// TwinCAT 3 PLC project PKE_Graz
// ProgramVersion: 3.1.4023.0
// libraries:
//   EfficientIO Communicator, * (EfficientIO)
//   Lynus Energy Basic, * (Lynus AG)
//   Lynus Energy ModbusTCP, * (Lynus AG)
//   Lynus Persistent Data V1, * (Lynus AG)
//   Lynus Standards, * (Lynus AG)
//   Tc2_ModbusSrv, * (Beckhoff Automation GmbH)
//   Tc2_Standard, * (Beckhoff Automation GmbH)
//   Tc2_System, * (Beckhoff Automation GmbH)
//   Tc2_Utilities, * (Beckhoff Automation GmbH)
//   Tc3_Module, * (Beckhoff Automation GmbH)
// project tree:
//   / FastTask.TcTTO, MiddleTask.TcTTO, SlowTask.TcTTO
//   FB/ FB_ModBus_100Reg_once_FC3.TcPOU, FB_ModBus_2Registers_FC3_T.TcPOU, F_DWORD_TO_FLOAT32.TcPOU
//   POUs/ prgComEffIO.TcPOU, PrgModbus.TcPOU, prgPersistent.TcPOU, prgRWEffIO.TcPOU, prgVarEffIO.TcPOU (not stored)
// real-time tasks:
//   TASK MiddleTask: cycle T#10ms, priority 20, ADS port 350
//   TASK FastTask: cycle T#5ms, priority 19, ADS port 351
//   TASK SlowTask: cycle T#20ms, priority 21, ADS port 352

CONFIGURATION PKE_Graz
    RESOURCE PLC ON TwinCAT3
        TASK FastTask(INTERVAL := T#5ms, PRIORITY := 19);
        TASK MiddleTask(INTERVAL := T#10ms, PRIORITY := 20);
        TASK SlowTask(INTERVAL := T#20ms, PRIORITY := 21);
        PROGRAM prgRWEffIO WITH FastTask : prgRWEffIO;
        PROGRAM prgVarEffIO WITH FastTask : prgVarEffIO;
        PROGRAM prgPersistent WITH MiddleTask : prgPersistent;
        PROGRAM PrgModbus WITH MiddleTask : PrgModbus;
        PROGRAM prgComEffIO WITH SlowTask : prgComEffIO;
    END_RESOURCE
END_CONFIGURATION

// ---- POUs/prgRWEffIO.TcPOU
PROGRAM prgRWEffIO
VAR
	fbRW1		: FB_ReadWrite_V2;
END_VAR

fbRW1(	eUploadType := eSelectDataUploadType.e_Change_Intervall5min,
		bBusy=> , 
		bError=> , 
		udiErrorCodeOut=> , 
		eErrorReadWrite_Out=> );

END_PROGRAM

// ---- POUs/prgPersistent.TcPOU
PROGRAM prgPersistent
VAR
	fbUSV		: FB_WritePersistentData_General;
	
	fb_Reboot		: NT_reboot;
	m_Reboot		: BOOL:=FALSE;
END_VAR

fbUSV(
	eSaveModeData:= eUSVSaveMode.eSaveEventBased, 
	bLoadPersistentDataOk=> , 
//	bPowerFailDetect=> , 
	bError=> , 
	bySaveProcess=> , 
	dwStorageLast24h=> , 
	udiErrorCode=> );
	
	
fb_Reboot(	netid := '',
			delay := 2,
			start := m_Reboot);

END_PROGRAM

// ---- POUs/PrgModbus.TcPOU
PROGRAM PrgModbus
VAR
	FB_Modbus: FB_ModBus_100Reg_once_FC3;
	fb_MB_WatchDog:FB_MBWriteSingleCoil ;
	fb_MB_Multi: FB_MBWriteRegs;

	str_IP	:STRING(20);
	
	i: INT;
	i_State: INT;
	ton_Wait_time: Ton;
	ton_TimeOut: ton;
	w_Array_Received: ARRAY [0..450] OF WORD;

	w_Array_Pol1_1: ARRAY [0..99] OF WORD;
	m_Pol1_1_ok: BOOL;
	w_Array_Pol1_2: ARRAY [0..99] OF WORD;
	m_Pol1_2_ok: BOOL;
	w_Array_Pol1_3: ARRAY [0..99] OF WORD;
	m_Pol1_3_ok: BOOL;
	w_Array_Pol1_4: ARRAY [0..99] OF WORD;
	m_Pol1_4_ok: BOOL;
	w_Array_Pol1_5: ARRAY [0..99] OF WORD;
	m_Pol1_5_ok: BOOL;
	w_Array_Pol1_6: ARRAY [0..99] OF WORD;
	m_Pol1_6_ok: BOOL;	
	int_Timeout: ARRAY [1..6] OF INT;
	
	real_EG_0_01_Testraum_Temp	: REAL;										//{#lynus.ag#()}
	real_EG_0_02_Werkstatt_Temp	: REAL;										//{#lynus.ag#()}
	real_EG_0_04_Buero1_Temp	: REAL;										//{#lynus.ag#()}
	real_EG_0_05_Buero2_Temp	: REAL;										//{#lynus.ag#()}
	real_EG_0_06_Leitung_Temp	: REAL;										//{#lynus.ag#()}
	real_EG_0_07_Service_Annahme_Temp	: REAL;								//{#lynus.ag#()}
	real_EG_0_08_Buero3_Temp	: REAL;										//{#lynus.ag#()}
	real_EG_0_09_Buero4_Temp	: REAL;										//{#lynus.ag#()}
	real_EG_0_10_Buero5_Temp	: REAL;										//{#lynus.ag#()}
	real_EG_0_11_Buero6_Temp	: REAL;										//{#lynus.ag#()}
	real_EG_0_12_Buero7_Temp	: REAL;										//{#lynus.ag#()}
	real_EG_0_13_Buero8_Temp	: REAL;										//{#lynus.ag#()}
	real_EG_0_14_Archiv_Temp	: REAL;										//{#lynus.ag#()}
	real_EG_0_20_WC_Damen_Beh_Temp	: REAL;									//{#lynus.ag#()}
	real_EG_0_23_CAD_Reserve_Temp	: REAL;									//{#lynus.ag#()}
	real_EG_0_24_CAD_Temp	: REAL;											//{#lynus.ag#()}
	real_EG_0_25_Reserve_Temp	: REAL;										//{#lynus.ag#()}
	real_EG_0_26_Buero9_Temp	: REAL;										//{#lynus.ag#()}
	real_EG_0_27_ErschliessungEGSued_Temp	: REAL;							//{#lynus.ag#()}
	real_EG_0_27_Teekueche_Temp	: REAL;										//{#lynus.ag#()}
	real_EG_0_28_Buero8_Temp	: REAL;										//{#lynus.ag#()}
	real_EG_0_29_Buero10_Temp	: REAL;										//{#lynus.ag#()}
	real_EG_0_30_Demo_Temp	: REAL;											//{#lynus.ag#()}
	real_EG_0_31_Buero11_Temp	: REAL;										//{#lynus.ag#()}
	real_EG_0_32_Buero12_GF_Temp	: REAL;									//{#lynus.ag#()}
	real_EG_0_33_Buero13_GF_Temp	: REAL;									//{#lynus.ag#()}
	real_EG_0_35_Buero14_Temp	: REAL;										//{#lynus.ag#()}
	real_EG_0_36_Buero15_Temp	: REAL;										//{#lynus.ag#()}
	real_EG_0_37_Buero16_Temp	: REAL;										//{#lynus.ag#()}
	real_EG_0_39_Buero17_Temp	: REAL;										//{#lynus.ag#()}
	real_EG_0_40_Besprechung_Temp	: REAL;									//{#lynus.ag#()}
	real_EG_0_42_WC_Beh_Temp	: REAL;										//{#lynus.ag#()}
	real_H_0_02_LagerPKE_Temp	: REAL;										//{#lynus.ag#()}
	real_H_00_03_Buero_LagerPKE_Temp	: Real;								//{#lynus.ag#()}
	real_OG1_1_01_Empfang_Temp	: REAL;										//{#lynus.ag#()}
	real_OG1_1_03_Buero1_Temp	: REAL;										//{#lynus.ag#()}
	real_OG1_1_04_Buero2_Temp	: REAL;										//{#lynus.ag#()}
	real_OG1_1_05_Buero3_Temp	: REAL;										//{#lynus.ag#()}
	real_OG1_1_06_Buero4_Temp	: REAL;										//{#lynus.ag#()}
	real_OG1_1_07_Buero_Besprechung_Temp	: REAL;							//{#lynus.ag#()}
	real_OG1_1_1_08_Plotter_Temp	: REAL;									//{#lynus.ag#()}
	real_OG1_1_04_WC_Herren_Temp	: REAL;									//{#lynus.ag#()}
	real_OG1_Serverraum_Temp	: REAL;										//{#lynus.ag#()}
	real_OG1_4_01_Empfang_Temp	: REAL;										//{#lynus.ag#()}
	real_OG1_4_03_Lager_Temp	: REAL;										//{#lynus.ag#()}
	real_OG1_4_04_Buero1_Temp	: REAL;										//{#lynus.ag#()}
	real_OG1_4_05_Buero2_Temp	: REAL;										//{#lynus.ag#()}
	real_OG1_4_06_Buero3_Temp	: REAL;										//{#lynus.ag#()}
	real_OG1_4_07_Buero4_Temp	: REAL;										//{#lynus.ag#()}
	real_OG1_4_08_Buero5_Temp	: REAL;										//{#lynus.ag#()}
	real_OG1_4_09_Buero6_Temp	: REAL;										//{#lynus.ag#()}
	real_OG1_4_10_AufenthaltKueche_Temp	: Real;								//{#lynus.ag#()}
	real_OG1_4_11_Besprechung_Temp	: REAL;									//{#lynus.ag#()}
	real_OG1_4_14_WC_Damen_Temp	: REAL;										//{#lynus.ag#()}
	real_OG1_2_03_Buero2_Temp	: REAL;										//{#lynus.ag#()}
	real_OG1_2_04_Besprechung_Temp	: REAL;									//{#lynus.ag#()}
	real_OG1_2_05_Server_VTOG2_Temp	: REAL;									//{#lynus.ag#()}
	real_OG1_2_06_Buero3_Temp	: REAL;										//{#lynus.ag#()}
	real_OG1_2_07_Buero4_Temp	: REAL;										//{#lynus.ag#()}
	real_OG1_3_xx_Besprechung_Temp	: REAL;									//{#lynus.ag#()}
	real_OG1_3_02_Buero1_Temp	: REAL;										//{#lynus.ag#()}
	real_OG1_3_03_Buero2_Temp	: REAL;										//{#lynus.ag#()}
	real_OG1_3_05_Server_Temp	: REAL;										//{#lynus.ag#()}
	real_OG1_3_06_Vorraum_WC_Temp	: REAL;									//{#lynus.ag#()}
	real_OG1_3_09_Empfang_Temp	: REAL;										//{#lynus.ag#()}
	real_OG1_3_10_Buero3_Temp	: REAL;										//{#lynus.ag#()}
	real_OG1_3_11_Buero4_Temp	: REAL;										//{#lynus.ag#()}
	real_H01_VL_Temp	: REAL;												//{#lynus.ag#()}
	real_H01_RL_Temp	: REAL;												//{#lynus.ag#()}
	real_H02_VL_Temp	: REAL;												//{#lynus.ag#()}
	real_H02_RL_Temp	: REAL;												//{#lynus.ag#()}
	real_H03_VL_Temp	: REAL;												//{#lynus.ag#()}
	real_H03_RL_Temp	: REAL;												//{#lynus.ag#()}
	real_H04_VL_Temp	: REAL;												//{#lynus.ag#()}
	real_H04_RL_Temp	: REAL;												//{#lynus.ag#()}
	real_H05_VL_Temp	: REAL;												//{#lynus.ag#()}
	real_H05_RL_Temp	: REAL;												//{#lynus.ag#()}
	real_H06_VL_Temp	: REAL;												//{#lynus.ag#()}
	real_H06_RL_Temp	: REAL;												//{#lynus.ag#()}
	real_SP_Schneider_H01_Temp_HZG	: REAL;									//{#lynus.ag#()}
	real_SP_Schneider_H02_Temp_HZG	: REAL;									//{#lynus.ag#()}
	real_SP_Schneider_H03_Temp_HZG	: REAL;									//{#lynus.ag#()}
	real_SP_Schneider_H04_Temp_HZG	: REAL;									//{#lynus.ag#()}
	real_SP_Schneider_H05_Temp_HZG	: REAL;									//{#lynus.ag#()}
	real_SP_Schneider_H06_Temp_HZG	: REAL;									//{#lynus.ag#()}
	real_SP_Schneider_H01_Temp_KLG	: REAL;									//{#lynus.ag#()}
	real_SP_Schneider_H02_Temp_KLG	: REAL;									//{#lynus.ag#()}
	real_SP_Schneider_H03_Temp_KLG	: REAL;									//{#lynus.ag#()}
	real_SP_Schneider_H04_Temp_KLG	: REAL;									//{#lynus.ag#()}
	real_SP_Schneider_H05_Temp_KLG	: REAL;									//{#lynus.ag#()}
	real_SP_Schneider_H06_Temp_KLG	: REAL;									//{#lynus.ag#()}
	real_L01_ZUL_Temp	: REAL;												//{#lynus.ag#()}
	real_L01_ABL_Temp	: REAL;												//{#lynus.ag#()}
	real_L01_AUL_Temp	: REAL;												//{#lynus.ag#()}
	real_L01_FOL_Temp	: REAL;												//{#lynus.ag#()}
	real_L01_SE_ZUL_Temp	: REAL;											//{#lynus.ag#()}
	real_L01_SW_Rot_WT	: REAL;												//{#lynus.ag#()}
	real_L01_SW_E_HZ_Reg	: REAL;											//{#lynus.ag#()}
	real_AT	: REAL;															//{#lynus.ag#()}
	real_SP_EfficientIO_H01_Temp_HZG	: Real;								//{#lynus.ag#()}
	real_SP_EfficientIO_H02_Temp_HZG	: Real;								//{#lynus.ag#()}
	real_SP_EfficientIO_H03_Temp_HZG	: Real;								//{#lynus.ag#()}
	real_SP_EfficientIO_H04_Temp_HZG	: Real;								//{#lynus.ag#()}
	real_SP_EfficientIO_H05_Temp_HZG	: Real;								//{#lynus.ag#()}
	real_SP_EfficientIO_H06_Temp_HZG	: Real;								//{#lynus.ag#()}
	real_SP_EfficientIO_H01_Temp_KLG	: Real;								//{#lynus.ag#()}
	real_SP_EfficientIO_H02_Temp_KLG	: Real;								//{#lynus.ag#()}
	real_SP_EfficientIO_H03_Temp_KLG	: Real;								//{#lynus.ag#()}
	real_SP_EfficientIO_H04_Temp_KLG	: Real;								//{#lynus.ag#()}
	real_SP_EfficientIO_H05_Temp_KLG	: Real;								//{#lynus.ag#()}
	real_SP_EfficientIO_H06_Temp_KLG	: Real;								//{#lynus.ag#()}
	real_SP_EfficientIO_H01_Temp_HZG_received	: REAL;				
	real_SP_EfficientIO_H02_Temp_HZG_received	: REAL;				
	real_SP_EfficientIO_H03_Temp_HZG_received	: REAL;				
	real_SP_EfficientIO_H04_Temp_HZG_received	: REAL;				
	real_SP_EfficientIO_H05_Temp_HZG_received	: REAL;				
	real_SP_EfficientIO_H06_Temp_HZG_received	: REAL;				
	real_SP_EfficientIO_H01_Temp_KLG_received	: REAL;				
	real_SP_EfficientIO_H02_Temp_KLG_received	: REAL;				
	real_SP_EfficientIO_H03_Temp_KLG_received	: REAL;				
	real_SP_EfficientIO_H04_Temp_KLG_received	: REAL;				
	real_SP_EfficientIO_H05_Temp_KLG_received	: REAL;				
	real_SP_EfficientIO_H06_Temp_KLG_received	: REAL;				
	usint_Betriebsart_H01	: USINT;										//{#lynus.ag#()}
	usint_Betriebsart_H02	: USINT;										//{#lynus.ag#()}
	usint_Betriebsart_H03	: USINT;										//{#lynus.ag#()}
	usint_Betriebsart_H04	: USINT;										//{#lynus.ag#()}
	usint_Betriebsart_H05	: USINT;										//{#lynus.ag#()}
	usint_Betriebsart_H06	: USINT;										//{#lynus.ag#()}
	m_Watchdog	: BOOL;														//{#lynus.ag#()}
	real_ZUL_errechnet_Schneider_Temp	: Real;								//{#lynus.ag#()}
	real_ZUL_errechnet_EfficientIO_Temp	: Real;								//{#lynus.ag#()}
	real_ZUL_errechnet_EfficientIO_Temp_received : REAL;
	FB_Convert_Real_to_Word:		 FB_CV_REAL_FLOAT_TO_WORD;
	f_trig_BussyWrite: f_trig;
	intArray_WriteError				: ARRAY[1..3] OF INT;		//error counter for each write command
	wArray_Data_To_Send				: ARRAY[1..40] OF WORD;		//word array to write 
	TON_HeartBeat2: Ton;
	TON_HeartBeat1: Ton;
	mEnable: BOOL;
	w_adress: WORD;
	nUnitID: BYTE;
	FB_2Reg :FB_ModBus_2Registers_FC3_T;

	ton_Wait2_time: TON;
	intArray_PollOk:  ARRAY [1..6] OF INT;
	intArray_WriteOk:  ARRAY [1..3] OF INT;

	m_Mode_Off_H01				: BOOL;									//{#lynus.ag#()}
	m_Mode_Heating_H01			: BOOL;									//{#lynus.ag#()}
	m_Mode_ReducedHeating_H01	: BOOL;									//{#lynus.ag#()}
	m_Mode_Frost_H01			: BOOL;									//{#lynus.ag#()}
	m_Mode_Cooling_H01			: BOOL;									//{#lynus.ag#()}
	m_Mode_ReducedCooling_H01	: BOOL;									//{#lynus.ag#()}

	m_Mode_Off_H02				: BOOL;									//{#lynus.ag#()}
	m_Mode_Heating_H02			: BOOL;									//{#lynus.ag#()}
	m_Mode_Frost_H02			: BOOL;									//{#lynus.ag#()}
	m_Mode_Cooling_H02			: BOOL;									//{#lynus.ag#()}

	m_Mode_Off_H03				: BOOL;									//{#lynus.ag#()}
	m_Mode_Heating_H03			: BOOL;									//{#lynus.ag#()}
	m_Mode_Frost_H03			: BOOL;									//{#lynus.ag#()}
	m_Mode_Cooling_H03			: BOOL;									//{#lynus.ag#()}

	m_Mode_Off_H04				: BOOL;									//{#lynus.ag#()}
	m_Mode_Heating_H04			: BOOL;									//{#lynus.ag#()}
	m_Mode_Frost_H04			: BOOL;									//{#lynus.ag#()}
	m_Mode_Cooling_H04			: BOOL;									//{#lynus.ag#()}

	m_Mode_Off_H05				: BOOL;									//{#lynus.ag#()}
	m_Mode_Heating_H05			: BOOL;									//{#lynus.ag#()}
	m_Mode_Frost_H05			: BOOL;									//{#lynus.ag#()}
	m_Mode_Cooling_H05			: BOOL;									//{#lynus.ag#()}

	m_Mode_Off_H06				: BOOL;									//{#lynus.ag#()}
	m_Mode_Heating_H06			: BOOL;									//{#lynus.ag#()}
	m_Mode_Frost_H06			: BOOL;									//{#lynus.ag#()}
	m_Mode_Cooling_H06			: BOOL;									//{#lynus.ag#()}

	
	
	int_HeartBeat					: INT;										//{#lynus.ag#()}
	byte_ErrorWarning				: BYTE;										//{#lynus.ag#()}
	m_EnergyOptimicingReady			: BOOL;										//{#lynus.ag#()}

	real_Power_H01				:REAL;									//{#lynus.ag#()}
	real_Power_H02				:REAL;									//{#lynus.ag#()}
	real_Power_H03				:REAL;									//{#lynus.ag#()}
	real_Power_H04				:REAL;									//{#lynus.ag#()}
	real_Power_H05				:REAL;									//{#lynus.ag#()}
	real_Power_H06				:REAL;									//{#lynus.ag#()}
	
	real_EnergyHeating_H01				:REAL;									//{#lynus.ag#()}
	real_EnergyHeating_H02				:REAL;									//{#lynus.ag#()}
	real_EnergyHeating_H03				:REAL;									//{#lynus.ag#()}
	real_EnergyHeating_H04				:REAL;									//{#lynus.ag#()}
	real_EnergyHeating_H05				:REAL;									//{#lynus.ag#()}
	real_EnergyHeating_H06				:REAL;									//{#lynus.ag#()}

	real_EnergyCooling_H01				:REAL;									//{#lynus.ag#()}
	real_EnergyCooling_H02				:REAL;									//{#lynus.ag#()}
	real_EnergyCooling_H03				:REAL;									//{#lynus.ag#()}
	real_EnergyCooling_H04				:REAL;									//{#lynus.ag#()}
	real_EnergyCooling_H05				:REAL;									//{#lynus.ag#()}
	real_EnergyCooling_H06				:REAL;									//{#lynus.ag#()}
	
	real_Power_HeatPump1				:REAL;									//{#lynus.ag#()}
	real_Power_HeatPump2				:REAL;									//{#lynus.ag#()}
	
	int_Count: INT;
END_VAR
VAR PERSISTENT
	m_EnableHeartbeat: BOOL;												//{#lynus.ag#()}
	m_Enbale_Write: BOOL:=TRUE;
END_VAR

// state maschine modbus
(*
FB_2Reg(
	m_Enable:= mEnable , 
	str_IPAdress:= '10.148.188.27', 
	w_Adress:= w_adress, 
	int_Divider:= 1, 
	n_UnitID:= nUnitID, 
	m_Float32Conversion:= , 
	m_PollSuccessful=> , 
	r_ReceivedValue=> , 
	udint_Error_ID=> );
*)

CASE i_State OF
	0: // wait state
		ton_Wait_time.IN := TRUE;
		IF ton_Wait_time.Q THEN
			ton_Wait_time.IN :=FALSE;
			i_State := 1;
		END_IF
	
	
	1: // Poll 1 Register 200 - 299
		FB_Modbus.m_Enable := TRUE;
		FB_Modbus.w_Adress := 199; //201;
		FB_Modbus.usint_Quantity := 100;
		
		ton_TimeOut.IN := TRUE;
		
		// wait for received values
		IF  FB_Modbus.m_PollSuccessful THEN
			FB_Modbus.m_Enable := FALSE;
			m_Pol1_1_ok := TRUE;			
			w_Array_Pol1_1 := FB_Modbus.w_Array_Received;
			FOR i:=0 TO FB_Modbus.usint_Quantity-1 BY 1 DO
				w_Array_Received[200+i] := w_Array_Pol1_1[i];
				w_Array_Pol1_1[i]:=0;
			END_FOR
			ton_TimeOut.IN := FALSE;
			i_State := 2;
		END_IF
		IF ton_TimeOut.Q THEN
			FB_Modbus.m_Enable := FALSE;
			ton_TimeOut.IN := FALSE;
			m_Pol1_1_ok := FALSE;			
			int_Timeout[1] := int_Timeout[1]+1;
			i_State := 2;
		END_IF
	
	2: // wait one cycle
		IF m_Pol1_1_ok THEN 
			m_Pol1_1_ok := FALSE;
			intArray_PollOk[1]:=intArray_PollOk[1]+1;
		END_IF
		i_State := 3;
		
	3: // Poll 2 Register 300 - 399
		FB_Modbus.m_Enable := TRUE;
		FB_Modbus.w_Adress := 299; //301;
		FB_Modbus.usint_Quantity := 100;
		
		ton_TimeOut.IN := TRUE;
		
		// wait for received values
		IF  FB_Modbus.m_PollSuccessful THEN
			FB_Modbus.m_Enable := FALSE;
			m_Pol1_2_ok := TRUE;
			w_Array_Pol1_2 := FB_Modbus.w_Array_Received;
			FOR i:=0 TO FB_Modbus.usint_Quantity-1 BY 1 DO
				w_Array_Received[300+i] := w_Array_Pol1_2[i];
				w_Array_Pol1_2[i]:=0;
			END_FOR
			ton_TimeOut.IN := FALSE;
			i_State := 4;
		END_IF
		IF ton_TimeOut.Q THEN
			FB_Modbus.m_Enable := FALSE;			
			ton_TimeOut.IN := FALSE;
			m_Pol1_2_ok := FALSE;
			int_Timeout[2] := int_Timeout[2]+1;
			i_State := 4;
		END_IF		
	
	4: // wait one cycle
		IF m_Pol1_2_ok THEN 
			m_Pol1_2_ok := FALSE;
			intArray_PollOk[2]:=intArray_PollOk[2]+1;
		END_IF		
		i_State := 5;
		
	5: // Poll 3 Register 400 - 426
		FB_Modbus.m_Enable := TRUE;
		FB_Modbus.w_Adress := 399; //401;
		FB_Modbus.usint_Quantity := 28;
		
		ton_TimeOut.IN := TRUE;
		
		// wait for received values
		IF  FB_Modbus.m_PollSuccessful THEN
			FB_Modbus.m_Enable := FALSE;
			m_Pol1_3_ok := TRUE;
			w_Array_Pol1_3 := FB_Modbus.w_Array_Received;
			FOR i:=0 TO FB_Modbus.usint_Quantity-1 BY 1 DO
				w_Array_Received[400+i] := w_Array_Pol1_3[i];
				w_Array_Pol1_3[i]:=0;
			END_FOR			
			ton_TimeOut.IN := FALSE;
			i_State := 6;
		END_IF
		IF ton_TimeOut.Q THEN
			FB_Modbus.m_Enable := FALSE;		
			ton_TimeOut.IN := FALSE;
			m_Pol1_3_ok := FALSE;
			int_Timeout[3] := int_Timeout[3]+1;
			i_State := 6;
		END_IF		

	6: // wait one cycle
		IF m_Pol1_3_ok THEN 
			m_Pol1_3_ok := FALSE;
			intArray_PollOk[3]:=intArray_PollOk[3]+1;
		END_IF		
		i_State := 7;
		
	7: // Poll 4 Register 432 - 436
		FB_Modbus.m_Enable := TRUE;
		FB_Modbus.w_Adress := 431; 
		FB_Modbus.usint_Quantity := 4;
		
		ton_TimeOut.IN := TRUE;
		
		// wait for received values
		IF  FB_Modbus.m_PollSuccessful THEN
			FB_Modbus.m_Enable := FALSE;
			m_Pol1_4_ok := TRUE;
			w_Array_Pol1_4 := FB_Modbus.w_Array_Received;
			FOR i:=0 TO FB_Modbus.usint_Quantity-1 BY 1 DO
				w_Array_Received[432+i] := w_Array_Pol1_4[i];
				w_Array_Pol1_4[i]:=0;
			END_FOR			
			ton_TimeOut.IN := FALSE;
			i_State := 8;
		END_IF
		IF ton_TimeOut.Q THEN
			FB_Modbus.m_Enable := FALSE;		
			ton_TimeOut.IN := FALSE;
			m_Pol1_4_ok := FALSE;
			int_Timeout[4] := int_Timeout[4]+1;
			i_State := 8;
		END_IF		
		
	8: // wait one cycle
		IF m_Pol1_4_ok THEN 
			m_Pol1_4_ok := FALSE;
			intArray_PollOk[4]:=intArray_PollOk[4]+1;
		END_IF		
		i_State := 9;
		
	9: // Poll 5 Register 1 - 99
		FB_Modbus.m_Enable := TRUE;
		FB_Modbus.w_Adress := 0; 
		FB_Modbus.usint_Quantity := 100;
		
		ton_TimeOut.IN := TRUE;
		
		// wait for received values
		IF  FB_Modbus.m_PollSuccessful THEN
			FB_Modbus.m_Enable := FALSE;
			m_Pol1_5_ok := TRUE;
			w_Array_Pol1_5 := FB_Modbus.w_Array_Received;
			FOR i:=0 TO FB_Modbus.usint_Quantity-1 BY 1 DO
				w_Array_Received[0+i] := w_Array_Pol1_5[i];
				w_Array_Pol1_5[i]:=0;
			END_FOR
			ton_TimeOut.IN := FALSE;
			i_State := 10;
		END_IF
		IF ton_TimeOut.Q THEN
			FB_Modbus.m_Enable := FALSE;			
			ton_TimeOut.IN := FALSE;
			m_Pol1_5_ok := FALSE;
			int_Timeout[5] := int_Timeout[5]+1;
			i_State := 10;
		END_IF		
	
	10: // wait one cycle
		IF m_Pol1_5_ok THEN 
			m_Pol1_5_ok := FALSE;
			intArray_PollOk[5]:=intArray_PollOk[5]+1;
		END_IF		
		i_State := 11;

	11: // Poll 6 Register 100 - 126
		FB_Modbus.m_Enable := TRUE;
		FB_Modbus.w_Adress := 100; 
		FB_Modbus.usint_Quantity := 26;
		
		ton_TimeOut.IN := TRUE;
		
		// wait for received values
		IF  FB_Modbus.m_PollSuccessful THEN
			FB_Modbus.m_Enable := FALSE;
			m_Pol1_6_ok := TRUE;
			w_Array_Pol1_6 := FB_Modbus.w_Array_Received;
			FOR i:=0 TO FB_Modbus.usint_Quantity-1 BY 1 DO
				w_Array_Received[99+i] := w_Array_Pol1_6[i];
				w_Array_Pol1_6[i]:=0;
			END_FOR
			ton_TimeOut.IN := FALSE;
			i_State := 12;
		END_IF
		IF ton_TimeOut.Q THEN
			FB_Modbus.m_Enable := FALSE;			
			ton_TimeOut.IN := FALSE;
			m_Pol1_6_ok := FALSE;
			int_Timeout[6] := int_Timeout[6]+1;
			i_State := 12;
		END_IF		
	
	12: // wait one cycle
		IF m_Pol1_6_ok THEN 
			m_Pol1_6_ok := FALSE;
			intArray_PollOk[6]:=intArray_PollOk[6]+1;
		END_IF		
		i_State := 18;
	
	18: // wait timer
		ton_Wait2_time.IN := TRUE;
		IF ton_Wait2_time.Q THEN
			ton_Wait2_time.IN :=FALSE;
			i_State :=19;
		END_IF

	19: // wait one cycle and prepare data
		IF m_Enbale_Write THEN
			// convert data for write

			FB_Convert_Real_to_Word(	rInputValue:= real_SP_EfficientIO_H01_Temp_HZG,
										eByteOrderForConvert := 1 ,
										wOutputValue_1 => wArray_Data_To_Send[1] ,
										wOutputValue_2 => wArray_Data_To_Send[2]);	
			FB_Convert_Real_to_Word(	rInputValue:= real_SP_EfficientIO_H02_Temp_HZG,
										eByteOrderForConvert := 1 ,
										wOutputValue_1 => wArray_Data_To_Send[3] ,
										wOutputValue_2 => wArray_Data_To_Send[4]);	
			FB_Convert_Real_to_Word(	rInputValue:= real_SP_EfficientIO_H03_Temp_HZG,
										eByteOrderForConvert := 1 ,
										wOutputValue_1 => wArray_Data_To_Send[5] ,
										wOutputValue_2 => wArray_Data_To_Send[6]);	
			FB_Convert_Real_to_Word(	rInputValue:= real_SP_EfficientIO_H04_Temp_HZG,
										eByteOrderForConvert := 1 ,
										wOutputValue_1 => wArray_Data_To_Send[7] ,
										wOutputValue_2 => wArray_Data_To_Send[8]);	
			FB_Convert_Real_to_Word(	rInputValue:= real_SP_EfficientIO_H05_Temp_HZG,
										eByteOrderForConvert := 1 ,
										wOutputValue_1 => wArray_Data_To_Send[9] ,
										wOutputValue_2 => wArray_Data_To_Send[10]);	
			FB_Convert_Real_to_Word(	rInputValue:= real_SP_EfficientIO_H06_Temp_HZG,
										eByteOrderForConvert := 1 ,
										wOutputValue_1 => wArray_Data_To_Send[11] ,
										wOutputValue_2 => wArray_Data_To_Send[12]);	
			FB_Convert_Real_to_Word(	rInputValue:= real_SP_EfficientIO_H01_Temp_KLG,
										eByteOrderForConvert := 1 ,
										wOutputValue_1 => wArray_Data_To_Send[13] ,
										wOutputValue_2 => wArray_Data_To_Send[14]);	
			FB_Convert_Real_to_Word(	rInputValue:= real_SP_EfficientIO_H02_Temp_KLG,
										eByteOrderForConvert := 1 ,
										wOutputValue_1 => wArray_Data_To_Send[15] ,
										wOutputValue_2 => wArray_Data_To_Send[16]);	
			FB_Convert_Real_to_Word(	rInputValue:= real_SP_EfficientIO_H03_Temp_KLG,
										eByteOrderForConvert := 1 ,
										wOutputValue_1 => wArray_Data_To_Send[17] ,
										wOutputValue_2 => wArray_Data_To_Send[18]);	
			FB_Convert_Real_to_Word(	rInputValue:= real_SP_EfficientIO_H04_Temp_KLG,
										eByteOrderForConvert := 1 ,
										wOutputValue_1 => wArray_Data_To_Send[19] ,
										wOutputValue_2 => wArray_Data_To_Send[20]);	
			FB_Convert_Real_to_Word(	rInputValue:= real_SP_EfficientIO_H05_Temp_KLG,
										eByteOrderForConvert := 1 ,
										wOutputValue_1 => wArray_Data_To_Send[21] ,
										wOutputValue_2 => wArray_Data_To_Send[22]);	
			FB_Convert_Real_to_Word(	rInputValue:= real_SP_EfficientIO_H06_Temp_KLG,
										eByteOrderForConvert := 1 ,
										wOutputValue_1 => wArray_Data_To_Send[23] ,
										wOutputValue_2 => wArray_Data_To_Send[24]);			
			FB_Convert_Real_to_Word(	rInputValue:= real_ZUL_errechnet_EfficientIO_Temp,
										eByteOrderForConvert := 1 ,
										wOutputValue_1 => wArray_Data_To_Send[25] ,
										wOutputValue_2 => wArray_Data_To_Send[26]);

			i_State := 20;
		ELSE	// Write not enabled
			i_State := 0;
		END_IF

	20: // write1 / Reg 398-421 
		
		fb_MB_Multi.bExecute := TRUE;
		fb_MB_Multi.nMBAddr := 397;
		fb_MB_Multi.nQuantity := 24;
		fb_MB_Multi.cbLength := WORD_TO_UDINT(fb_MB_Multi.nQuantity*2);
		fb_MB_Multi.pSrcAddr := ADR(wArray_Data_To_Send[1]);
		
		ton_TimeOut.IN := TRUE;
		// wait for write successfull
		f_trig_BussyWrite (CLK := fb_MB_Multi.bBusy);
		
		IF f_trig_BussyWrite.Q OR ton_TimeOut.Q THEN
			fb_MB_Multi.bExecute := FALSE;
			ton_TimeOut.IN := FALSE;
			IF NOT fb_MB_Multi.bError THEN
				intArray_WriteOk[1] := intArray_WriteOk[1]+1;
				i_State := i_State+1;
			ELSIF fb_MB_Multi.bError OR ton_TimeOut.Q THEN
				intArray_WriteError[1] := intArray_WriteError[1]+1;
				i_State := i_State+1;
			END_IF
		END_IF
		
	21: // wait state
		ton_Wait_time.IN := TRUE;
		IF ton_Wait_time.Q THEN
			ton_Wait_time.IN :=FALSE;
			i_State := 30;
		END_IF	

	30: // write2 / Reg 434 
		
		fb_MB_Multi.bExecute := TRUE;
		fb_MB_Multi.nMBAddr := 433;
		fb_MB_Multi.nQuantity := 2;
		fb_MB_Multi.cbLength := WORD_TO_UDINT(fb_MB_Multi.nQuantity*2);
		fb_MB_Multi.pSrcAddr := ADR(wArray_Data_To_Send[25]);
		
		ton_TimeOut.IN := TRUE;
		// wait for write successfull
		f_trig_BussyWrite (CLK := fb_MB_Multi.bBusy);
		
		IF f_trig_BussyWrite.Q OR ton_TimeOut.Q THEN
			fb_MB_Multi.bExecute := FALSE;
			ton_TimeOut.IN := FALSE;
			IF NOT fb_MB_Multi.bError THEN
				intArray_WriteOk[2] := intArray_WriteOk[2]+1;
				i_State := i_State+1;
			ELSIF fb_MB_Multi.bError OR ton_TimeOut.Q THEN
				intArray_WriteError[2] := intArray_WriteError[2]+1;
				i_State := i_State+1;
			END_IF
		END_IF
		
	31: // wait state
		ton_Wait_time.IN := TRUE;
		IF ton_Wait_time.Q THEN
			ton_Wait_time.IN :=FALSE;
			i_State := 40;
		END_IF
	
	40: // write single coil / Watchdog / Reg 429 

		fb_MB_WatchDog.bExecute := TRUE;
		fb_MB_WatchDog.nMBAddr := 429;
		
		IF m_Watchdog THEN
			fb_MB_WatchDog.nValue := 16#FF00;
		ELSE
			fb_MB_WatchDog.nValue := 16#0000;
		END_IF
				
		ton_TimeOut.IN := TRUE;
		// wait for write successfull
		f_trig_BussyWrite (CLK := fb_MB_WatchDog.bBusy);
		
		IF f_trig_BussyWrite.Q OR ton_TimeOut.Q THEN
			fb_MB_WatchDog.bExecute := FALSE;
			ton_TimeOut.IN := FALSE;
			IF NOT fb_MB_WatchDog.bError THEN
				intArray_WriteOk[3] := intArray_WriteOk[3]+1;
				i_State := i_State+1;
			ELSIF fb_MB_WatchDog.bError OR ton_TimeOut.Q THEN
				intArray_WriteError[3] := intArray_WriteError[3]+1;
				i_State := i_State+1;
			END_IF
		END_IF
		
	41: // wait state
		ton_Wait_time.IN := TRUE;
		IF ton_Wait_time.Q THEN
			ton_Wait_time.IN :=FALSE;
			i_State := 100;
		END_IF



	100: // wait one cycle and start from the beginning
		i_State := 0;
		
		
END_CASE


IF m_EnableHeartbeat THEN
	m_Enbale_Write :=TRUE;
	IF TON_HeartBeat1.Q THEN
		m_Watchdog:=1;		
	ELSE
		m_Watchdog:=0;		
	END_IF
ELSE
	m_Enbale_Write :=FALSE;
END_IF

TON_HeartBeat1(	IN:= TRUE AND NOT TON_HeartBeat2.Q ,
		PT:= T#15S,
		Q=> );
TON_HeartBeat2(	IN:= TON_HeartBeat1.Q,
		PT:= T#15S);
		
		
ton_Wait_time(PT:=T#500MS);
ton_Wait2_time(PT:=T#2S);
ton_TimeOut(PT:=T#10S);  // must be higher then t#5s because internal timeout timer
str_IP := '10.148.188.27';

FB_Modbus(
	m_Enable:= , 
	str_IPAdress:= str_IP, 
	w_Adress:= , 
	usint_Quantity:= ,
	nUnitID := 1, 
	m_PollSuccessful=> , 
	w_Array_Received=> , 
	udint_Error_ID=> );

fb_MB_WatchDog(
	sIPAddr:= str_IP, 
	nTCPPort:= 502 , 
	nUnitID:= 1, 
	nMBAddr:= , 
	nValue:= , 
	bExecute:= , 
	tTimeout:=  T#5S, 
	bBusy=> , 
	bError=> , 
	nErrId=> );
	
fb_MB_Multi(
	sIPAddr:= str_IP, 
	nTCPPort:= 502, 
	nUnitID:= 1, 
	nQuantity:= , 
	nMBAddr:= , 
	cbLength:= , 
	pSrcAddr:= , 
	bExecute:= , 
	tTimeout:= T#5S , 
	bBusy=> , 
	bError=> , 
	nErrId=> );

	
// copy modbus data if poll is successfull	
IF m_Pol1_1_ok THEN
	real_EG_0_01_Testraum_Temp				:=  F_DWORD_TO_FLOAT32(dwInput  :=  WORD_TO_DWORD(w_Array_Received[200]) + 16#10000 * WORD_TO_DWORD(w_Array_Received[201])); 
	real_EG_0_02_Werkstatt_Temp 			:=  F_DWORD_TO_FLOAT32(dwInput  :=  WORD_TO_DWORD(w_Array_Received[202]) + 16#10000 * WORD_TO_DWORD(w_Array_Received[203])); 
	real_EG_0_04_Buero1_Temp 				:=  F_DWORD_TO_FLOAT32(dwInput  :=  WORD_TO_DWORD(w_Array_Received[204]) + 16#10000 * WORD_TO_DWORD(w_Array_Received[205])); 
	real_EG_0_05_Buero2_Temp 				:=  F_DWORD_TO_FLOAT32(dwInput  :=  WORD_TO_DWORD(w_Array_Received[206]) + 16#10000 * WORD_TO_DWORD(w_Array_Received[207])); 
	real_EG_0_06_Leitung_Temp 				:=  F_DWORD_TO_FLOAT32(dwInput  :=  WORD_TO_DWORD(w_Array_Received[208]) + 16#10000 * WORD_TO_DWORD(w_Array_Received[209])); 
	real_EG_0_07_Service_Annahme_Temp 		:=  F_DWORD_TO_FLOAT32(dwInput  :=  WORD_TO_DWORD(w_Array_Received[210]) + 16#10000 * WORD_TO_DWORD(w_Array_Received[211])); 
	real_EG_0_08_Buero3_Temp 				:=  F_DWORD_TO_FLOAT32(dwInput  :=  WORD_TO_DWORD(w_Array_Received[212]) + 16#10000 * WORD_TO_DWORD(w_Array_Received[213])); 
	real_EG_0_09_Buero4_Temp 				:=  F_DWORD_TO_FLOAT32(dwInput  :=  WORD_TO_DWORD(w_Array_Received[214]) + 16#10000 * WORD_TO_DWORD(w_Array_Received[215])); 
	real_EG_0_10_Buero5_Temp 				:=  F_DWORD_TO_FLOAT32(dwInput  :=  WORD_TO_DWORD(w_Array_Received[216]) + 16#10000 * WORD_TO_DWORD(w_Array_Received[217])); 
	real_EG_0_11_Buero6_Temp 				:=  F_DWORD_TO_FLOAT32(dwInput  :=  WORD_TO_DWORD(w_Array_Received[218]) + 16#10000 * WORD_TO_DWORD(w_Array_Received[219])); 
	real_EG_0_12_Buero7_Temp 				:=  F_DWORD_TO_FLOAT32(dwInput  :=  WORD_TO_DWORD(w_Array_Received[220]) + 16#10000 * WORD_TO_DWORD(w_Array_Received[221])); 
	real_EG_0_13_Buero8_Temp 				:=  F_DWORD_TO_FLOAT32(dwInput  :=  WORD_TO_DWORD(w_Array_Received[222]) + 16#10000 * WORD_TO_DWORD(w_Array_Received[223])); 
	real_EG_0_14_Archiv_Temp 				:=  F_DWORD_TO_FLOAT32(dwInput  :=  WORD_TO_DWORD(w_Array_Received[224]) + 16#10000 * WORD_TO_DWORD(w_Array_Received[225])); 
	real_EG_0_20_WC_Damen_Beh_Temp 			:=  F_DWORD_TO_FLOAT32(dwInput  :=  WORD_TO_DWORD(w_Array_Received[226]) + 16#10000 * WORD_TO_DWORD(w_Array_Received[227])); 
	real_EG_0_23_CAD_Reserve_Temp 			:=  F_DWORD_TO_FLOAT32(dwInput  :=  WORD_TO_DWORD(w_Array_Received[228]) + 16#10000 * WORD_TO_DWORD(w_Array_Received[229])); 
	real_EG_0_24_CAD_Temp 					:=  F_DWORD_TO_FLOAT32(dwInput  :=  WORD_TO_DWORD(w_Array_Received[230]) + 16#10000 * WORD_TO_DWORD(w_Array_Received[231])); 
	real_EG_0_25_Reserve_Temp 				:=  F_DWORD_TO_FLOAT32(dwInput  :=  WORD_TO_DWORD(w_Array_Received[232]) + 16#10000 * WORD_TO_DWORD(w_Array_Received[233])); 
	real_EG_0_26_Buero9_Temp 				:=  F_DWORD_TO_FLOAT32(dwInput  :=  WORD_TO_DWORD(w_Array_Received[234]) + 16#10000 * WORD_TO_DWORD(w_Array_Received[235])); 
	real_EG_0_27_ErschliessungEGSued_Temp 	:=  F_DWORD_TO_FLOAT32(dwInput  :=  WORD_TO_DWORD(w_Array_Received[236]) + 16#10000 * WORD_TO_DWORD(w_Array_Received[237])); 
	real_EG_0_27_Teekueche_Temp 			:=  F_DWORD_TO_FLOAT32(dwInput  :=  WORD_TO_DWORD(w_Array_Received[238]) + 16#10000 * WORD_TO_DWORD(w_Array_Received[239])); 
	real_EG_0_28_Buero8_Temp 				:=  F_DWORD_TO_FLOAT32(dwInput  :=  WORD_TO_DWORD(w_Array_Received[240]) + 16#10000 * WORD_TO_DWORD(w_Array_Received[241])); 
	real_EG_0_29_Buero10_Temp 				:=  F_DWORD_TO_FLOAT32(dwInput  :=  WORD_TO_DWORD(w_Array_Received[242]) + 16#10000 * WORD_TO_DWORD(w_Array_Received[243])); 
	real_EG_0_30_Demo_Temp 					:=  F_DWORD_TO_FLOAT32(dwInput  :=  WORD_TO_DWORD(w_Array_Received[244]) + 16#10000 * WORD_TO_DWORD(w_Array_Received[245])); 
	real_EG_0_31_Buero11_Temp 				:=  F_DWORD_TO_FLOAT32(dwInput  :=  WORD_TO_DWORD(w_Array_Received[246]) + 16#10000 * WORD_TO_DWORD(w_Array_Received[247])); 
	real_EG_0_32_Buero12_GF_Temp 			:=  F_DWORD_TO_FLOAT32(dwInput  :=  WORD_TO_DWORD(w_Array_Received[248]) + 16#10000 * WORD_TO_DWORD(w_Array_Received[249])); 
	real_EG_0_33_Buero13_GF_Temp 			:=  F_DWORD_TO_FLOAT32(dwInput  :=  WORD_TO_DWORD(w_Array_Received[250]) + 16#10000 * WORD_TO_DWORD(w_Array_Received[251])); 
	real_EG_0_35_Buero14_Temp 				:=  F_DWORD_TO_FLOAT32(dwInput  :=  WORD_TO_DWORD(w_Array_Received[252]) + 16#10000 * WORD_TO_DWORD(w_Array_Received[253])); 
	real_EG_0_36_Buero15_Temp 				:=  F_DWORD_TO_FLOAT32(dwInput  :=  WORD_TO_DWORD(w_Array_Received[254]) + 16#10000 * WORD_TO_DWORD(w_Array_Received[255])); 
	real_EG_0_37_Buero16_Temp 				:=  F_DWORD_TO_FLOAT32(dwInput  :=  WORD_TO_DWORD(w_Array_Received[256]) + 16#10000 * WORD_TO_DWORD(w_Array_Received[257])); 
	real_EG_0_39_Buero17_Temp 				:=  F_DWORD_TO_FLOAT32(dwInput  :=  WORD_TO_DWORD(w_Array_Received[258]) + 16#10000 * WORD_TO_DWORD(w_Array_Received[259])); 
	real_EG_0_40_Besprechung_Temp 			:=  F_DWORD_TO_FLOAT32(dwInput  :=  WORD_TO_DWORD(w_Array_Received[260]) + 16#10000 * WORD_TO_DWORD(w_Array_Received[261])); 
	real_EG_0_42_WC_Beh_Temp 				:=  F_DWORD_TO_FLOAT32(dwInput  :=  WORD_TO_DWORD(w_Array_Received[262]) + 16#10000 * WORD_TO_DWORD(w_Array_Received[263])); 
	real_H_0_02_LagerPKE_Temp 				:=  F_DWORD_TO_FLOAT32(dwInput  :=  WORD_TO_DWORD(w_Array_Received[264]) + 16#10000 * WORD_TO_DWORD(w_Array_Received[265])); 
	real_H_00_03_Buero_LagerPKE_Temp 		:=  F_DWORD_TO_FLOAT32(dwInput  :=  WORD_TO_DWORD(w_Array_Received[266]) + 16#10000 * WORD_TO_DWORD(w_Array_Received[267])); 
	real_OG1_1_01_Empfang_Temp 				:=  F_DWORD_TO_FLOAT32(dwInput  :=  WORD_TO_DWORD(w_Array_Received[268]) + 16#10000 * WORD_TO_DWORD(w_Array_Received[269])); 
	real_OG1_1_03_Buero1_Temp 				:=  F_DWORD_TO_FLOAT32(dwInput  :=  WORD_TO_DWORD(w_Array_Received[270]) + 16#10000 * WORD_TO_DWORD(w_Array_Received[271])); 
	real_OG1_1_04_Buero2_Temp 				:=  F_DWORD_TO_FLOAT32(dwInput  :=  WORD_TO_DWORD(w_Array_Received[272]) + 16#10000 * WORD_TO_DWORD(w_Array_Received[273])); 
	real_OG1_1_05_Buero3_Temp 				:=  F_DWORD_TO_FLOAT32(dwInput  :=  WORD_TO_DWORD(w_Array_Received[274]) + 16#10000 * WORD_TO_DWORD(w_Array_Received[275])); 
	real_OG1_1_06_Buero4_Temp 				:=  F_DWORD_TO_FLOAT32(dwInput  :=  WORD_TO_DWORD(w_Array_Received[276]) + 16#10000 * WORD_TO_DWORD(w_Array_Received[277])); 
	real_OG1_1_07_Buero_Besprechung_Temp 	:=  F_DWORD_TO_FLOAT32(dwInput  :=  WORD_TO_DWORD(w_Array_Received[278]) + 16#10000 * WORD_TO_DWORD(w_Array_Received[279])); 
	real_OG1_1_1_08_Plotter_Temp 			:=  F_DWORD_TO_FLOAT32(dwInput  :=  WORD_TO_DWORD(w_Array_Received[280]) + 16#10000 * WORD_TO_DWORD(w_Array_Received[281])); 
	real_OG1_1_04_WC_Herren_Temp			:=  F_DWORD_TO_FLOAT32(dwInput  :=  WORD_TO_DWORD(w_Array_Received[282]) + 16#10000 * WORD_TO_DWORD(w_Array_Received[283])); 
	real_OG1_Serverraum_Temp 				:=  F_DWORD_TO_FLOAT32(dwInput  :=  WORD_TO_DWORD(w_Array_Received[284]) + 16#10000 * WORD_TO_DWORD(w_Array_Received[285])); 
	real_OG1_4_01_Empfang_Temp 				:=  F_DWORD_TO_FLOAT32(dwInput  :=  WORD_TO_DWORD(w_Array_Received[286]) + 16#10000 * WORD_TO_DWORD(w_Array_Received[287])); 
	real_OG1_4_03_Lager_Temp 				:=  F_DWORD_TO_FLOAT32(dwInput  :=  WORD_TO_DWORD(w_Array_Received[288]) + 16#10000 * WORD_TO_DWORD(w_Array_Received[289])); 
	real_OG1_4_04_Buero1_Temp 				:=  F_DWORD_TO_FLOAT32(dwInput  :=  WORD_TO_DWORD(w_Array_Received[290]) + 16#10000 * WORD_TO_DWORD(w_Array_Received[291])); 
	real_OG1_4_05_Buero2_Temp				:=  F_DWORD_TO_FLOAT32(dwInput  :=  WORD_TO_DWORD(w_Array_Received[292]) + 16#10000 * WORD_TO_DWORD(w_Array_Received[293])); 
	real_OG1_4_06_Buero3_Temp 				:=  F_DWORD_TO_FLOAT32(dwInput  :=  WORD_TO_DWORD(w_Array_Received[294]) + 16#10000 * WORD_TO_DWORD(w_Array_Received[295])); 
	real_OG1_4_07_Buero4_Temp 				:=  F_DWORD_TO_FLOAT32(dwInput  :=  WORD_TO_DWORD(w_Array_Received[296]) + 16#10000 * WORD_TO_DWORD(w_Array_Received[297])); 
	real_OG1_4_08_Buero5_Temp 				:=  F_DWORD_TO_FLOAT32(dwInput  :=  WORD_TO_DWORD(w_Array_Received[298]) + 16#10000 * WORD_TO_DWORD(w_Array_Received[299])); 
END_IF

IF m_Pol1_2_ok THEN
	real_OG1_4_09_Buero6_Temp				:=  F_DWORD_TO_FLOAT32(dwInput  :=  WORD_TO_DWORD(w_Array_Received[300]) + 16#10000 * WORD_TO_DWORD(w_Array_Received[301])); 
	real_OG1_4_10_AufenthaltKueche_Temp 	:=  F_DWORD_TO_FLOAT32(dwInput  :=  WORD_TO_DWORD(w_Array_Received[302]) + 16#10000 * WORD_TO_DWORD(w_Array_Received[303])); 
	real_OG1_4_11_Besprechung_Temp 			:=  F_DWORD_TO_FLOAT32(dwInput  :=  WORD_TO_DWORD(w_Array_Received[304]) + 16#10000 * WORD_TO_DWORD(w_Array_Received[305])); 
	real_OG1_4_14_WC_Damen_Temp 			:=  F_DWORD_TO_FLOAT32(dwInput  :=  WORD_TO_DWORD(w_Array_Received[306]) + 16#10000 * WORD_TO_DWORD(w_Array_Received[307])); 
	real_OG1_2_03_Buero2_Temp 				:=  F_DWORD_TO_FLOAT32(dwInput  :=  WORD_TO_DWORD(w_Array_Received[308]) + 16#10000 * WORD_TO_DWORD(w_Array_Received[309])); 
	real_OG1_2_04_Besprechung_Temp 			:=  F_DWORD_TO_FLOAT32(dwInput  :=  WORD_TO_DWORD(w_Array_Received[310]) + 16#10000 * WORD_TO_DWORD(w_Array_Received[311])); 
	real_OG1_2_05_Server_VTOG2_Temp 		:=  F_DWORD_TO_FLOAT32(dwInput  :=  WORD_TO_DWORD(w_Array_Received[312]) + 16#10000 * WORD_TO_DWORD(w_Array_Received[313])); 
	real_OG1_2_06_Buero3_Temp 				:=  F_DWORD_TO_FLOAT32(dwInput  :=  WORD_TO_DWORD(w_Array_Received[314]) + 16#10000 * WORD_TO_DWORD(w_Array_Received[315])); 
	real_OG1_2_07_Buero4_Temp 				:=  F_DWORD_TO_FLOAT32(dwInput  :=  WORD_TO_DWORD(w_Array_Received[316]) + 16#10000 * WORD_TO_DWORD(w_Array_Received[317])); 
	real_OG1_3_xx_Besprechung_Temp 			:=  F_DWORD_TO_FLOAT32(dwInput  :=  WORD_TO_DWORD(w_Array_Received[318]) + 16#10000 * WORD_TO_DWORD(w_Array_Received[319])); 
	real_OG1_3_02_Buero1_Temp 				:=  F_DWORD_TO_FLOAT32(dwInput  :=  WORD_TO_DWORD(w_Array_Received[320]) + 16#10000 * WORD_TO_DWORD(w_Array_Received[321])); 
	real_OG1_3_03_Buero2_Temp 				:=  F_DWORD_TO_FLOAT32(dwInput  :=  WORD_TO_DWORD(w_Array_Received[322]) + 16#10000 * WORD_TO_DWORD(w_Array_Received[323])); 
	real_OG1_3_05_Server_Temp 				:=  F_DWORD_TO_FLOAT32(dwInput  :=  WORD_TO_DWORD(w_Array_Received[324]) + 16#10000 * WORD_TO_DWORD(w_Array_Received[325])); 
	real_OG1_3_06_Vorraum_WC_Temp 			:=  F_DWORD_TO_FLOAT32(dwInput  :=  WORD_TO_DWORD(w_Array_Received[326]) + 16#10000 * WORD_TO_DWORD(w_Array_Received[327])); 
	real_OG1_3_09_Empfang_Temp 				:=  F_DWORD_TO_FLOAT32(dwInput  :=  WORD_TO_DWORD(w_Array_Received[328]) + 16#10000 * WORD_TO_DWORD(w_Array_Received[329])); 
	real_OG1_3_10_Buero3_Temp 				:=  F_DWORD_TO_FLOAT32(dwInput  :=  WORD_TO_DWORD(w_Array_Received[330]) + 16#10000 * WORD_TO_DWORD(w_Array_Received[331])); 
	real_OG1_3_11_Buero4_Temp 				:=  F_DWORD_TO_FLOAT32(dwInput  :=  WORD_TO_DWORD(w_Array_Received[332]) + 16#10000 * WORD_TO_DWORD(w_Array_Received[333])); 
	real_H01_VL_Temp 						:=  F_DWORD_TO_FLOAT32(dwInput  :=  WORD_TO_DWORD(w_Array_Received[334]) + 16#10000 * WORD_TO_DWORD(w_Array_Received[335])); 
	real_H01_RL_Temp 						:=  F_DWORD_TO_FLOAT32(dwInput  :=  WORD_TO_DWORD(w_Array_Received[336]) + 16#10000 * WORD_TO_DWORD(w_Array_Received[337])); 
	real_H02_VL_Temp						:=  F_DWORD_TO_FLOAT32(dwInput  :=  WORD_TO_DWORD(w_Array_Received[338]) + 16#10000 * WORD_TO_DWORD(w_Array_Received[339])); 
	real_H02_RL_Temp 						:=  F_DWORD_TO_FLOAT32(dwInput  :=  WORD_TO_DWORD(w_Array_Received[340]) + 16#10000 * WORD_TO_DWORD(w_Array_Received[341])); 
	real_H03_VL_Temp 						:=  F_DWORD_TO_FLOAT32(dwInput  :=  WORD_TO_DWORD(w_Array_Received[342]) + 16#10000 * WORD_TO_DWORD(w_Array_Received[343])); 
	real_H03_RL_Temp 						:=  F_DWORD_TO_FLOAT32(dwInput  :=  WORD_TO_DWORD(w_Array_Received[344]) + 16#10000 * WORD_TO_DWORD(w_Array_Received[345])); 
	real_H04_VL_Temp 						:=  F_DWORD_TO_FLOAT32(dwInput  :=  WORD_TO_DWORD(w_Array_Received[346]) + 16#10000 * WORD_TO_DWORD(w_Array_Received[347])); 
	real_H04_RL_Temp 						:=  F_DWORD_TO_FLOAT32(dwInput  :=  WORD_TO_DWORD(w_Array_Received[348]) + 16#10000 * WORD_TO_DWORD(w_Array_Received[349])); 
	real_H05_VL_Temp 						:=  F_DWORD_TO_FLOAT32(dwInput  :=  WORD_TO_DWORD(w_Array_Received[350]) + 16#10000 * WORD_TO_DWORD(w_Array_Received[351])); 
	real_H05_RL_Temp 						:=  F_DWORD_TO_FLOAT32(dwInput  :=  WORD_TO_DWORD(w_Array_Received[352]) + 16#10000 * WORD_TO_DWORD(w_Array_Received[353])); 
	real_H06_VL_Temp 						:=  F_DWORD_TO_FLOAT32(dwInput  :=  WORD_TO_DWORD(w_Array_Received[354]) + 16#10000 * WORD_TO_DWORD(w_Array_Received[355])); 
	real_H06_RL_Temp 						:=  F_DWORD_TO_FLOAT32(dwInput  :=  WORD_TO_DWORD(w_Array_Received[356]) + 16#10000 * WORD_TO_DWORD(w_Array_Received[357])); 
	real_SP_Schneider_H01_Temp_HZG 			:=  F_DWORD_TO_FLOAT32(dwInput  :=  WORD_TO_DWORD(w_Array_Received[358]) + 16#10000 * WORD_TO_DWORD(w_Array_Received[359])); 
	real_SP_Schneider_H02_Temp_HZG 			:=  F_DWORD_TO_FLOAT32(dwInput  :=  WORD_TO_DWORD(w_Array_Received[360]) + 16#10000 * WORD_TO_DWORD(w_Array_Received[361])); 
	real_SP_Schneider_H03_Temp_HZG 			:=  F_DWORD_TO_FLOAT32(dwInput  :=  WORD_TO_DWORD(w_Array_Received[362]) + 16#10000 * WORD_TO_DWORD(w_Array_Received[363])); 
	real_SP_Schneider_H04_Temp_HZG 			:=  F_DWORD_TO_FLOAT32(dwInput  :=  WORD_TO_DWORD(w_Array_Received[364]) + 16#10000 * WORD_TO_DWORD(w_Array_Received[365])); 
	real_SP_Schneider_H05_Temp_HZG 			:=  F_DWORD_TO_FLOAT32(dwInput  :=  WORD_TO_DWORD(w_Array_Received[366]) + 16#10000 * WORD_TO_DWORD(w_Array_Received[367])); 
	real_SP_Schneider_H06_Temp_HZG 			:=  F_DWORD_TO_FLOAT32(dwInput  :=  WORD_TO_DWORD(w_Array_Received[368]) + 16#10000 * WORD_TO_DWORD(w_Array_Received[369])); 
	real_SP_Schneider_H01_Temp_KLG 			:=  F_DWORD_TO_FLOAT32(dwInput  :=  WORD_TO_DWORD(w_Array_Received[370]) + 16#10000 * WORD_TO_DWORD(w_Array_Received[371])); 
	real_SP_Schneider_H02_Temp_KLG 			:=  F_DWORD_TO_FLOAT32(dwInput  :=  WORD_TO_DWORD(w_Array_Received[372]) + 16#10000 * WORD_TO_DWORD(w_Array_Received[373])); 
	real_SP_Schneider_H03_Temp_KLG 			:=  F_DWORD_TO_FLOAT32(dwInput  :=  WORD_TO_DWORD(w_Array_Received[374]) + 16#10000 * WORD_TO_DWORD(w_Array_Received[375])); 
	real_SP_Schneider_H04_Temp_KLG 			:=  F_DWORD_TO_FLOAT32(dwInput  :=  WORD_TO_DWORD(w_Array_Received[376]) + 16#10000 * WORD_TO_DWORD(w_Array_Received[377])); 
	real_SP_Schneider_H05_Temp_KLG 			:=  F_DWORD_TO_FLOAT32(dwInput  :=  WORD_TO_DWORD(w_Array_Received[378]) + 16#10000 * WORD_TO_DWORD(w_Array_Received[379])); 
	real_SP_Schneider_H06_Temp_KLG 			:=  F_DWORD_TO_FLOAT32(dwInput  :=  WORD_TO_DWORD(w_Array_Received[380]) + 16#10000 * WORD_TO_DWORD(w_Array_Received[381])); 
	real_L01_ZUL_Temp 						:=  F_DWORD_TO_FLOAT32(dwInput  :=  WORD_TO_DWORD(w_Array_Received[382]) + 16#10000 * WORD_TO_DWORD(w_Array_Received[383])); 
	real_L01_ABL_Temp 						:=  F_DWORD_TO_FLOAT32(dwInput  :=  WORD_TO_DWORD(w_Array_Received[384]) + 16#10000 * WORD_TO_DWORD(w_Array_Received[385])); 
	real_L01_AUL_Temp 						:=  F_DWORD_TO_FLOAT32(dwInput  :=  WORD_TO_DWORD(w_Array_Received[386]) + 16#10000 * WORD_TO_DWORD(w_Array_Received[387])); 
	real_L01_FOL_Temp 						:=  F_DWORD_TO_FLOAT32(dwInput  :=  WORD_TO_DWORD(w_Array_Received[388]) + 16#10000 * WORD_TO_DWORD(w_Array_Received[389])); 
	real_L01_SE_ZUL_Temp 					:=  F_DWORD_TO_FLOAT32(dwInput  :=  WORD_TO_DWORD(w_Array_Received[390]) + 16#10000 * WORD_TO_DWORD(w_Array_Received[391])); 
	real_L01_SW_Rot_WT 						:=  F_DWORD_TO_FLOAT32(dwInput  :=  WORD_TO_DWORD(w_Array_Received[392]) + 16#10000 * WORD_TO_DWORD(w_Array_Received[393])); 
	real_L01_SW_E_HZ_Reg 					:=  F_DWORD_TO_FLOAT32(dwInput  :=  WORD_TO_DWORD(w_Array_Received[394]) + 16#10000 * WORD_TO_DWORD(w_Array_Received[395])); 
	real_AT 								:=  F_DWORD_TO_FLOAT32(dwInput  :=  WORD_TO_DWORD(w_Array_Received[396]) + 16#10000 * WORD_TO_DWORD(w_Array_Received[397])); 
	real_SP_EfficientIO_H01_Temp_HZG_received 		:=  F_DWORD_TO_FLOAT32(dwInput  :=  WORD_TO_DWORD(w_Array_Received[398]) + 16#10000 * WORD_TO_DWORD(w_Array_Received[399])); 
END_IF
	
IF m_Pol1_3_ok THEN
	real_SP_EfficientIO_H02_Temp_HZG_received		:=  F_DWORD_TO_FLOAT32(dwInput  :=  WORD_TO_DWORD(w_Array_Received[400]) + 16#10000 * WORD_TO_DWORD(w_Array_Received[401])); 
	real_SP_EfficientIO_H03_Temp_HZG_received 		:=  F_DWORD_TO_FLOAT32(dwInput  :=  WORD_TO_DWORD(w_Array_Received[402]) + 16#10000 * WORD_TO_DWORD(w_Array_Received[403])); 
	real_SP_EfficientIO_H04_Temp_HZG_received 		:=  F_DWORD_TO_FLOAT32(dwInput  :=  WORD_TO_DWORD(w_Array_Received[404]) + 16#10000 * WORD_TO_DWORD(w_Array_Received[405])); 
	real_SP_EfficientIO_H05_Temp_HZG_received		:=  F_DWORD_TO_FLOAT32(dwInput  :=  WORD_TO_DWORD(w_Array_Received[406]) + 16#10000 * WORD_TO_DWORD(w_Array_Received[407])); 
	real_SP_EfficientIO_H06_Temp_HZG_received 		:=  F_DWORD_TO_FLOAT32(dwInput  :=  WORD_TO_DWORD(w_Array_Received[408]) + 16#10000 * WORD_TO_DWORD(w_Array_Received[409])); 
	real_SP_EfficientIO_H01_Temp_KLG_received 		:=  F_DWORD_TO_FLOAT32(dwInput  :=  WORD_TO_DWORD(w_Array_Received[410]) + 16#10000 * WORD_TO_DWORD(w_Array_Received[411])); 
	real_SP_EfficientIO_H02_Temp_KLG_received 		:=  F_DWORD_TO_FLOAT32(dwInput  :=  WORD_TO_DWORD(w_Array_Received[412]) + 16#10000 * WORD_TO_DWORD(w_Array_Received[413])); 
	real_SP_EfficientIO_H03_Temp_KLG_received 		:=  F_DWORD_TO_FLOAT32(dwInput  :=  WORD_TO_DWORD(w_Array_Received[414]) + 16#10000 * WORD_TO_DWORD(w_Array_Received[415])); 
	real_SP_EfficientIO_H04_Temp_KLG_received 		:=  F_DWORD_TO_FLOAT32(dwInput  :=  WORD_TO_DWORD(w_Array_Received[416]) + 16#10000 * WORD_TO_DWORD(w_Array_Received[417])); 
	real_SP_EfficientIO_H05_Temp_KLG_received		:=  F_DWORD_TO_FLOAT32(dwInput  :=  WORD_TO_DWORD(w_Array_Received[418]) + 16#10000 * WORD_TO_DWORD(w_Array_Received[419])); 
	real_SP_EfficientIO_H06_Temp_KLG_received 		:=  F_DWORD_TO_FLOAT32(dwInput  :=  WORD_TO_DWORD(w_Array_Received[420]) + 16#10000 * WORD_TO_DWORD(w_Array_Received[421])); 
	usint_Betriebsart_H01					:=  WORD_TO_USINT(w_Array_Received[422]); 
	usint_Betriebsart_H02 					:=  WORD_TO_USINT(w_Array_Received[423]); 
	usint_Betriebsart_H03  					:=  WORD_TO_USINT(w_Array_Received[424]);
	usint_Betriebsart_H04  					:=  WORD_TO_USINT(w_Array_Received[425]);
	usint_Betriebsart_H05  					:=  WORD_TO_USINT(w_Array_Received[426]);
	usint_Betriebsart_H06  					:=  WORD_TO_USINT(w_Array_Received[427]);
//	m_Watchdog 								:=  w_Array_Received[430].0; 
END_IF
IF m_Pol1_4_ok THEN
	real_ZUL_errechnet_Schneider_Temp 		:=  F_DWORD_TO_FLOAT32(dwInput  :=  WORD_TO_DWORD(w_Array_Received[432]) + 16#10000 * WORD_TO_DWORD(w_Array_Received[433])); 
	real_ZUL_errechnet_EfficientIO_Temp_received 	:=  F_DWORD_TO_FLOAT32(dwInput  :=  WORD_TO_DWORD(w_Array_Received[434]) + 16#10000 * WORD_TO_DWORD(w_Array_Received[435])); 
END_IF

IF m_Pol1_5_ok THEN
	int_Count :=-1;
	real_Power_H01 			:=  F_DWORD_TO_FLOAT32(dwInput  :=  WORD_TO_DWORD(w_Array_Received[3+int_Count]) + 16#10000 * WORD_TO_DWORD(w_Array_Received[4+int_Count])); 
	real_EnergyCooling_H01	:=  F_DWORD_TO_FLOAT32(dwInput  :=  WORD_TO_DWORD(w_Array_Received[5+int_Count]) + 16#10000 * WORD_TO_DWORD(w_Array_Received[6+int_Count])); 
	real_EnergyHeating_H01	:=  F_DWORD_TO_FLOAT32(dwInput  :=  WORD_TO_DWORD(w_Array_Received[7+int_Count]) + 16#10000 * WORD_TO_DWORD(w_Array_Received[8+int_Count]));
	int_Count :=7;
	real_Power_H02 			:=  F_DWORD_TO_FLOAT32(dwInput  :=  WORD_TO_DWORD(w_Array_Received[3+int_Count]) + 16#10000 * WORD_TO_DWORD(w_Array_Received[4+int_Count])); 
	real_EnergyCooling_H02	:=  F_DWORD_TO_FLOAT32(dwInput  :=  WORD_TO_DWORD(w_Array_Received[5+int_Count]) + 16#10000 * WORD_TO_DWORD(w_Array_Received[6+int_Count])); 
	real_EnergyHeating_H02	:=  F_DWORD_TO_FLOAT32(dwInput  :=  WORD_TO_DWORD(w_Array_Received[7+int_Count]) + 16#10000 * WORD_TO_DWORD(w_Array_Received[8+int_Count]));
	int_Count :=15;
	real_Power_H03 			:=  F_DWORD_TO_FLOAT32(dwInput  :=  WORD_TO_DWORD(w_Array_Received[3+int_Count]) + 16#10000 * WORD_TO_DWORD(w_Array_Received[4+int_Count])); 
	real_EnergyCooling_H03	:=  F_DWORD_TO_FLOAT32(dwInput  :=  WORD_TO_DWORD(w_Array_Received[5+int_Count]) + 16#10000 * WORD_TO_DWORD(w_Array_Received[6+int_Count])); 
	real_EnergyHeating_H03	:=  F_DWORD_TO_FLOAT32(dwInput  :=  WORD_TO_DWORD(w_Array_Received[7+int_Count]) + 16#10000 * WORD_TO_DWORD(w_Array_Received[8+int_Count]));
	int_Count :=23;
	real_Power_H04 			:=  F_DWORD_TO_FLOAT32(dwInput  :=  WORD_TO_DWORD(w_Array_Received[3+int_Count]) + 16#10000 * WORD_TO_DWORD(w_Array_Received[4+int_Count])); 
	real_EnergyCooling_H04	:=  F_DWORD_TO_FLOAT32(dwInput  :=  WORD_TO_DWORD(w_Array_Received[5+int_Count]) + 16#10000 * WORD_TO_DWORD(w_Array_Received[6+int_Count])); 
	real_EnergyHeating_H04	:=  F_DWORD_TO_FLOAT32(dwInput  :=  WORD_TO_DWORD(w_Array_Received[7+int_Count]) + 16#10000 * WORD_TO_DWORD(w_Array_Received[8+int_Count]));
	int_Count :=31;
	real_Power_H05 			:=  F_DWORD_TO_FLOAT32(dwInput  :=  WORD_TO_DWORD(w_Array_Received[3+int_Count]) + 16#10000 * WORD_TO_DWORD(w_Array_Received[4+int_Count])); 
	real_EnergyCooling_H05	:=  F_DWORD_TO_FLOAT32(dwInput  :=  WORD_TO_DWORD(w_Array_Received[5+int_Count]) + 16#10000 * WORD_TO_DWORD(w_Array_Received[6+int_Count])); 
	real_EnergyHeating_H05	:=  F_DWORD_TO_FLOAT32(dwInput  :=  WORD_TO_DWORD(w_Array_Received[7+int_Count]) + 16#10000 * WORD_TO_DWORD(w_Array_Received[8+int_Count]));	
	int_Count :=39;
	real_Power_H06 			:=  F_DWORD_TO_FLOAT32(dwInput  :=  WORD_TO_DWORD(w_Array_Received[3+int_Count]) + 16#10000 * WORD_TO_DWORD(w_Array_Received[4+int_Count])); 
	real_EnergyCooling_H06	:=  F_DWORD_TO_FLOAT32(dwInput  :=  WORD_TO_DWORD(w_Array_Received[5+int_Count]) + 16#10000 * WORD_TO_DWORD(w_Array_Received[6+int_Count])); 
	real_EnergyHeating_H06	:=  F_DWORD_TO_FLOAT32(dwInput  :=  WORD_TO_DWORD(w_Array_Received[7+int_Count]) + 16#10000 * WORD_TO_DWORD(w_Array_Received[8+int_Count]));
END_IF
IF m_Pol1_6_ok THEN
	real_Power_HeatPump1	:=  F_DWORD_TO_FLOAT32(dwInput  :=  WORD_TO_DWORD(w_Array_Received[105]) + 16#10000 * WORD_TO_DWORD(w_Array_Received[106])); 
	real_Power_HeatPump2	:=  F_DWORD_TO_FLOAT32(dwInput  :=  WORD_TO_DWORD(w_Array_Received[109]) + 16#10000 * WORD_TO_DWORD(w_Array_Received[110])); 
END_IF

m_Mode_Off_H01 				:= FALSE;
m_Mode_Heating_H01			:= FALSE;
m_Mode_Frost_H01			:= FALSE;
m_Mode_Cooling_H01			:= FALSE;
CASE usint_Betriebsart_H01 OF
	0: m_Mode_Off_H01 				:= TRUE;
	1,2: m_Mode_Heating_H01			:= TRUE;
	3: m_Mode_Frost_H01				:= TRUE;
	4,5: m_Mode_Cooling_H01			:= TRUE;
END_CASE

m_Mode_Off_H02 				:= FALSE;
m_Mode_Heating_H02			:= FALSE;
m_Mode_Frost_H02			:= FALSE;
m_Mode_Cooling_H02			:= FALSE;
CASE usint_Betriebsart_H02 OF
	0: m_Mode_Off_H02 				:= TRUE;
	1,2: m_Mode_Heating_H02			:= TRUE;
	3: m_Mode_Frost_H02				:= TRUE;
	4,5: m_Mode_Cooling_H02			:= TRUE;
END_CASE

m_Mode_Off_H03 				:= FALSE;
m_Mode_Heating_H03			:= FALSE;
m_Mode_Frost_H03			:= FALSE;
m_Mode_Cooling_H03			:= FALSE;
CASE usint_Betriebsart_H03 OF
	0: m_Mode_Off_H03 				:= TRUE;
	1,2: m_Mode_Heating_H03			:= TRUE;
	3: m_Mode_Frost_H03				:= TRUE;
	4,5: m_Mode_Cooling_H03			:= TRUE;
END_CASE

m_Mode_Off_H04 				:= FALSE;
m_Mode_Heating_H04			:= FALSE;
m_Mode_Frost_H04			:= FALSE;
m_Mode_Cooling_H04			:= FALSE;
CASE usint_Betriebsart_H04 OF
	0: m_Mode_Off_H04 				:= TRUE;
	1,2: m_Mode_Heating_H04			:= TRUE;
	3: m_Mode_Frost_H04				:= TRUE;
	4,5: m_Mode_Cooling_H04			:= TRUE;
END_CASE

m_Mode_Off_H05 				:= FALSE;
m_Mode_Heating_H05			:= FALSE;
m_Mode_Frost_H05			:= FALSE;
m_Mode_Cooling_H05			:= FALSE;
CASE usint_Betriebsart_H05 OF
	0: m_Mode_Off_H05 				:= TRUE;
	1,2: m_Mode_Heating_H05			:= TRUE;
	3: m_Mode_Frost_H05				:= TRUE;
	4,5: m_Mode_Cooling_H05			:= TRUE;
END_CASE

m_Mode_Off_H06 				:= FALSE;
m_Mode_Heating_H06			:= FALSE;
m_Mode_Frost_H06			:= FALSE;
m_Mode_Cooling_H06			:= FALSE;
CASE usint_Betriebsart_H06 OF
	0: m_Mode_Off_H06 				:= TRUE;
	1,2: m_Mode_Heating_H06			:= TRUE;
	3: m_Mode_Frost_H06				:= TRUE;
	4,5: m_Mode_Cooling_H06			:= TRUE;
END_CASE

END_PROGRAM

// ---- FB/FB_ModBus_100Reg_once_FC3.TcPOU
FUNCTION_BLOCK FB_ModBus_100Reg_once_FC3
VAR_INPUT PERSISTENT
	m_Enable					: BOOL;						// rising edge, read out once
	str_IPAdress				: STRING(15);				// IP Adress of the meter
	w_Adress					: WORD;						// modbus adress
	usint_Quantity				: USINT;					// Number of Words to get polled, max 100
	nUnitID						: BYTE:=255;				// Unit ID, default 255
END_VAR
VAR_OUTPUT
	m_PollSuccessful			: BOOL;						//Poll succesfull		
	w_Array_Received			: ARRAY[0..99] OF WORD;		// received data
	udint_Error_ID				: UDINT;					// ERR ID FB_MBReadRegs
END_VAR
VAR
	
	timer_TimeOut				: TON;						//Timer for Timeout MB Read
	
	iStateModbusRead			: INT;						//State machine for read out Data over Modbus RTU
	
	fbMBRead_FC3				: FB_MBReadRegs  ;		//Modbus Read Function (FC3)
	
	rtrig_PEnable				: r_trig;					//Internal positive Edge	
	iStateModbusError			: INT;						//State machine for error out Data over Modbus TCP/IP	
	
	FPError_FC_3				: R_TRIG;					//Internal positive Edge
	
	arrBuffer_FC3				: ARRAY[1..100] OF WORD;		//Buffer with Data from FC3
	
	timer_Connection_ok			: TON;
	int_Data_Received			: INT;
	
	m_MBTCPError				: BOOL;
	
	int_Data_Received_old		: INT;
	
	timer_Connection_ok_TOF	: TOF;
	
	fbConvertWordToDword		: FB_CV_WORD_TO_DWORD;			//Convert Word to Dword
	
	m_Poll_ok: BOOL;
	
	int_TimeoutError: INT;
	int_FC3Error: INT;

	timer_Delay: Ton;
	i: INT;
END_VAR

(*	{attribute 'hide'}--------------------------------------------------------------------------------------------Limits-------------------------------------------------------------------------------------*)

w_Adress := LIMIT(0,w_Adress,32767);
usint_Quantity := LIMIT(1,usint_Quantity,100);

(*--------------------------------------------------------------------------------------------State Machine Read--------------------------------------------------------------------------------------*)


//Timeout Timer is dissabled when the Init Step is aktiv or the function is not enabled
IF iStateModbusRead = 0 OR NOT m_Enable THEN 
	timer_Timeout.IN := FALSE; 
END_IF
timer_Timeout(IN:= , PT:= T#5S, Q=> , ET=> );


CASE iStateModbusRead OF

	0://Init Step 
		fbMBRead_FC3.bExecute := FALSE;
		m_Poll_ok:=FALSE;
		timer_Delay.IN := FALSE;
		int_Data_Received:=0;
		rtrig_PEnable(clk := m_Enable);
		IF rtrig_PEnable.Q THEN
			i:=i+1;
			iStateModbusRead := 1;
		END_IF
		
	1://read the required registers
		//Start Read
		fbMBRead_FC3.nQuantity := usint_Quantity;
		fbMBRead_FC3.nMBAddr := w_Adress;
		fbMBRead_FC3.bExecute := TRUE;
		fbMBRead_FC3.nUnitID := nUnitID;
		timer_Timeout.IN := TRUE;
		IF fbMBRead_FC3.bBusy THEN 
			timer_Delay.IN := TRUE; 
		END_IF

		//Wait for Delay, copy Data and then next step
		IF NOT fbMBRead_FC3.bBusy AND NOT fbMBRead_FC3.bError AND timer_Delay.Q THEN
			timer_Delay.IN := FALSE;
			m_Poll_ok:=TRUE;
			int_Data_Received:=int_Data_Received+1;
			m_MBTCPError := FALSE; 
			
			w_Array_Received := arrBuffer_FC3;
			
			
			//Go to Next Step
			timer_Timeout.IN := FALSE;
			fbMBRead_FC3.bExecute := FALSE;
			iStateModbusRead := 3;
		END_IF	

		//Error or Timeout
		IF FPError_FC_3.Q THEN 
			fbMBRead_FC3.bExecute := FALSE;
			timer_Delay.IN := FALSE;
			iStateModbusError := 300;
			int_FC3Error := int_FC3Error+1;
		ELSIF timer_Timeout.Q THEN  
			fbMBRead_FC3.bExecute := FALSE;
			timer_Delay.IN := FALSE;
			timer_Timeout.IN := FALSE; 	
			iStateModbusError := 300;
			int_TimeoutError := int_TimeoutError+1;
		END_IF
		
	
	3://Wait and go to step 0
		
		iStateModbusRead := 0;
				
		//Error on Master, changes on Inputs or Timeout
		IF timer_Timeout.Q THEN 
			iStateModbusError := 300; 
		END_IF
	
END_CASE




(*------------------------------------------------------------------Error and Warning----------------------------------------------------------------------------*)	
 
timer_Connection_ok			(In:=int_Data_Received<>int_Data_Received_old,PT:=T#10S);
timer_Connection_ok_TOF		(In:=NOT(int_Data_Received<>int_Data_Received_old) AND int_Data_Received>3 ,PT:=T#20S);
//Timer for Delay
timer_Delay(IN:= , PT:= T#50MS, Q=> , ET=> );

int_Data_Received_old:=int_Data_Received;
m_PollSuccessful:=m_Poll_ok ;

(*------------------------------------------------------------------------------------------Modbus TCP Functions---------------------------------------------------------------------------------------------*)

fbMBRead_FC3(	sIPAddr:= str_IPAdress, 
				nTCPPort:= 502,
				cbLength:= usint_Quantity*2 , //SIZEOF(arrBuffer_FC3), 
				pDestAddr:= ADR(arrBuffer_FC3), 
				tTimeout:= T#10S,
				nErrId => udint_Error_ID);

FPError_FC_3(CLK:= fbMBRead_FC3.bError, Q=> );		

(*------------------------------------------------------------------------------------------State Machine Error---------------------------------------------------------------------------------------------*)	

CASE iStateModbusError OF
	
	300://Error

		fbMBRead_FC3.bExecute := FALSE;
		m_MBTCPError := TRUE; 		
		m_Poll_ok:=FALSE;
		int_Data_Received:=0;
		//Restart from new with the Read out part after an Error
		iStateModbusRead := 0;	
		iStateModbusError := 0;
							
END_CASE

END_FUNCTION_BLOCK

// ---- FB/FB_ModBus_2Registers_FC3_T.TcPOU
FUNCTION_BLOCK FB_ModBus_2Registers_FC3_T
VAR_INPUT PERSISTENT
	m_Enable					: BOOL;						//Enable the Fuctionblock and his logic
	str_IPAdress				: STRING(15);				//IP Adress of the meter
	w_Adress					: WORD;						//modbus adress
	int_Divider					: INT;						//Devider of the received data
	n_UnitID					: BYTE:=255;				// dentification number of a serial sub-network device. If a device is addressed directly via TCP/IP, this value must be 16#FF / 255
	m_Float32Conversion			: BOOL;						// receives value in Float 32 / real format
END_VAR
VAR_OUTPUT
	m_PollSuccessful			: BOOL;						//Poll succesfull		
	r_ReceivedValue				: REAL;						//Received Value
	udint_Error_ID				: UDINT;					// ERR ID FB_MBReadRegs
END_VAR
VAR
	{attribute 'hide'}
	timer_Delay					: TON;						//Timer for Delay between Requests
	{attribute 'hide'}
	timer_DelayStart			: TON;						//Timer to start the state machine with Delay after enabling or after the system ist restartet
	{attribute 'hide'}
	timer_TimeOut				: TON;						//Timer for Timeout MB Read
	{attribute 'hide'}
	iStateModbusRead			: INT;						//State machine for read out Data over Modbus RTU
	{attribute 'hide'}
	fbMBRead_FC3				: FB_MBReadRegs ;		//Modbus Read Function (FC3)
	{attribute 'hide'}
	ftrig_PEnable				: f_trig;					//Internal positive Edge
	{attribute 'hide'}
	iStateModbusError			: INT;						//State machine for error out Data over Modbus TCP/IP	
	{attribute 'hide'}
	FPError_FC_3				: R_TRIG;					//Internal positive Edge
	{attribute 'hide'}
	arrBuffer_FC3				: ARRAY[1..2] OF WORD;		//Buffer with Data from FC3
	{attribute 'hide'}
	timer_Connection_ok			: TON;
	int_Data_Received			: INT;
	{attribute 'hide'}
	m_MBTCPError				: BOOL;
	{attribute 'hide'}
	int_Data_Received_old		: INT;
	{attribute 'hide'}
	timer_Connection_ok_TOF	: TOF;
	{attribute 'hide'}
	fbConvertWordToDword		: FB_CV_WORD_TO_DWORD;			//Convert Word to Dword
	{attribute 'hide'}
	usintSign					: USINT;						// converstion dword to real	
	{attribute 'hide'}
	intExponent					: INT;							// converstion dword to real
	{attribute 'hide'}
	realMantisse				: REAL;							// converstion dword to real
	{attribute 'hide'}
	m_Poll_ok: BOOL;
	{attribute 'hide'}
	timer_Wait: Ton;
	int_TimeoutError: INT;
	int_FC3Error: INT;
END_VAR

(*--------------------------------------------------------------------------------------------Limits-------------------------------------------------------------------------------------*)

w_Adress := LIMIT(0,w_Adress,65535);
int_Divider := LIMIT(1,int_Divider,32767);
	
(*--------------------------------------------------------------------------------------------State Machine Read--------------------------------------------------------------------------------------*)

//Timer for Delay
timer_Delay(IN:= , PT:= T#50MS, Q=> , ET=> );

//Timeout Timer is dissabled when the Init Step is aktiv or the function is not enabled
IF iStateModbusRead = 0 OR NOT m_Enable THEN 
	timer_Timeout.IN := FALSE; 
END_IF
timer_Timeout(IN:= , PT:= T#1S, Q=> , ET=> );

//Enable with Delay that not all sockets have to be created at the same time
timer_DelayStart(IN:= m_Enable, PT:= T#1S, Q=> , ET=> );
ftrig_PEnable(CLK:= timer_DelayStart.Q, Q=> );

IF ftrig_PEnable.Q AND iStateModbusRead = 0 THEN 
	iStateModbusRead := 1; 
END_IF		
		
//Not Enabled
IF NOT m_Enable THEN 
	iStateModbusRead := 0; 
	iStateModbusError := 0; 
END_IF		
		
CASE iStateModbusRead OF

	0://Init Step 
		timer_Delay.IN := FALSE;
		fbMBRead_FC3.bExecute := FALSE;
		m_Poll_ok:=FALSE;
		int_Data_Received:=0;
	
		iStateModbusRead := 1;
	
	1://read the required registers
		//Start Read
		fbMBRead_FC3.nQuantity := 2;
		fbMBRead_FC3.nMBAddr := w_Adress;
		fbMBRead_FC3.bExecute := TRUE;
		fbMBRead_FC3.nUnitID := n_UnitID;
		timer_Timeout.IN := TRUE;
		IF fbMBRead_FC3.bBusy THEN 
			timer_Delay.IN := TRUE; 
		END_IF
		
		//Wait for Delay, copy Data and then next step
		IF NOT fbMBRead_FC3.bBusy AND NOT fbMBRead_FC3.bError AND timer_Delay.Q THEN
			m_Poll_ok:=TRUE;
			int_Data_Received:=int_Data_Received+1;
			m_MBTCPError := FALSE; 
			// convert received data
			IF m_Float32Conversion THEN
		//		fbConvertWordToDword(wInputValue_1:= arrBuffer_FC3[1], wInputValue_2:= arrBuffer_FC3[2], eByteOrderForConvert:= eByteOrder.eLittleEndian , dwOutputValue=> );
				fbConvertWordToDword(wInputValue_1:= arrBuffer_FC3[1], wInputValue_2:= arrBuffer_FC3[2], eByteOrderForConvert:= 1 , dwOutputValue=> );
				(* Sign *)
				usintSign:=BOOL_TO_USINT(fbConvertWordToDword.dwOutputValue.31);
				(* Exponent *)
				intExponent:=DWORD_TO_INT(SHR(fbConvertWordToDword.dwOutputValue,23) AND 16#FF);
				(* Mantisse *)
				realMantisse:=DWORD_TO_REAL(fbConvertWordToDword.dwOutputValue AND 16#7FFFFF);
				(* Result *)
				r_ReceivedValue := LREAL_TO_REAL((EXPT((-1),usintSign) * (1+realMantisse/8388608) * EXPT(2,intExponent-127))/int_Divider);
			ELSE
				fbConvertWordToDword(wInputValue_1:= arrBuffer_FC3[2], wInputValue_2:= arrBuffer_FC3[1], eByteOrderForConvert:= eByteOrder.eLittleEndian , dwOutputValue=> );
				r_ReceivedValue := DINT_TO_REAL(fbConvertWordToDword.dwOutputValue)/int_Divider;
			END_IF
			
			//Go to Next Step
			timer_Timeout.IN := FALSE;
			fbMBRead_FC3.bExecute := FALSE;
			timer_Delay.IN := FALSE;		
			iStateModbusRead := 3;
		END_IF	

		//Error or Timeout
		IF FPError_FC_3.Q THEN 
			iStateModbusError := 300;
			int_FC3Error := int_FC3Error+1;
		ELSIF timer_Timeout.Q THEN 
			timer_Timeout.IN := FALSE; 	  	
			iStateModbusError := 300;
			int_TimeoutError := int_TimeoutError+1;
		END_IF
		
	
	3://Wait and go to step 1
		//1 because 0 is the Init Step for Read
		timer_Wait.IN := TRUE;
		
		IF timer_Wait.Q = TRUE THEN
			iStateModbusRead := 1;
			timer_Wait.IN :=FALSE;
		END_IF

			
		
		//Error on Master, changes on Inputs or Timeout
		IF timer_Timeout.Q THEN 
			iStateModbusError := 300; 
		END_IF
	
END_CASE

(* wait timer*)

timer_Wait(PT:=T#3S);


(*------------------------------------------------------------------Error and Warning----------------------------------------------------------------------------*)	
 
timer_Connection_ok			(In:=int_Data_Received<>int_Data_Received_old,PT:=T#10S);
timer_Connection_ok_TOF		(In:=NOT(int_Data_Received<>int_Data_Received_old) AND int_Data_Received>3 ,PT:=T#20S);
int_Data_Received_old:=int_Data_Received;
m_PollSuccessful:=NOT timer_Connection_ok.Q AND timer_Connection_ok_TOF.Q ;

(*------------------------------------------------------------------------------------------Modbus TCP Functions---------------------------------------------------------------------------------------------*)

fbMBRead_FC3(	sIPAddr:= str_IPAdress, 
				nTCPPort:= 502,
				cbLength:= SIZEOF(arrBuffer_FC3), 
				pDestAddr:= ADR(arrBuffer_FC3), 
				tTimeout:= T#10S,
				nErrId => udint_Error_ID);

FPError_FC_3(CLK:= fbMBRead_FC3.  bError, Q=> );		

(*------------------------------------------------------------------------------------------State Machine Error---------------------------------------------------------------------------------------------*)	

CASE iStateModbusError OF
	
	300://Error
		timer_Wait.IN :=TRUE;
		timer_Delay.IN := FALSE;
		fbMBRead_FC3.bExecute := FALSE;
		m_MBTCPError := TRUE; 		
		m_Poll_ok:=FALSE;
		int_Data_Received:=0;
				//Restart from new with the Read out part after an Error
		IF timer_Wait.Q = TRUE THEN
			iStateModbusRead := 0;	
			iStateModbusError := 0;
			timer_Wait.IN :=FALSE;
			timer_Timeout.IN := FALSE;
		END_IF		
							
END_CASE

END_FUNCTION_BLOCK

// ---- FB/F_DWORD_TO_FLOAT32.TcPOU
FUNCTION F_DWORD_TO_FLOAT32 : REAL
VAR_INPUT
	dwInput: DWORD;
END_VAR
VAR
	realSign: REAL;
	realExponent: REAL;
	realMantisse: REAL;
END_VAR

(* Sign *)
realSign:=BOOL_TO_REAL(dwInput.31);

(* Exponent *)
realExponent:=SHR(dwInput,23) AND 16#FF;

(* Mantisse *)
realMantisse:=dwInput AND 16#7FFFFF;

(* Result *)
F_DWORD_TO_FLOAT32:=EXPT((-1),realSign)*(1+realMantisse/8388608)*EXPT(2,realExponent-127);

(*if both register are 0*)
IF dwInput=0 THEN
	F_DWORD_TO_FLOAT32 :=0;
END_IF

END_FUNCTION

// ---- POUs/prgComEffIO.TcPOU
PROGRAM prgComEffIO
VAR
	fbCom		: FB_MqttCommunicator_V2;
END_VAR

fbCom(
	bConnect				:= TRUE,
	strAuthKey				:= 'EIO08031879806', 
	sUserName				:= '825f07c4-bbac-469f-beae-0c4ad006bf93', 
	sUserPassword			:= 'b1111145-4452-4020-8dff-f640d68312f3', 
	eSavePositionCertificate:= eSavePositionOnPLC.ePostionC, 
	bConnected=> , 
	bError=> , 
	hrErrorCode=> , 
	eConnectionState=> , 
	eErrorMessage_Out=> );

END_PROGRAM
